// TIA Portal project "XSFW_TIA05601_A5" (V15)

(* hardware
DEVICE "S7-1200 station_1"  S7-1200 Station
   slot 0: "Rack_0"  S7-1200 Rack  Rack  V1.0
   slot 1: "PLC_1"  CPU 1214C DC/DC/DC  6ES7 214-1AG40-0XB0  V4.2
DEVICE "Dispositivo GSD_1"  GSD.Device.PN
   slot 0: "Rack"  Rack  V1.0
   slot 0: "SINAMICS-S120-CU320-2PN"  SINAMICS S120/S150 CU320-2 PN V4.7  6SL3 040-1MA01-0AAx  V4.70
      slot 0: "SINAMICS S120/S150 CU320-2 PN V4.7"  SINAMICS S120/S150 CU320-2 PN V4.7
      slot 1: "PN-IO"  PN-IO
         slot 1: "Puerto 1"  Port 1
         slot 2: "Puerto 2"  Port 2
   slot 1: "DO Control Unit_1"  DO Control Unit
      slot 0: "Punto de acceso a módulo"  Module Access Point
      slot 1: "sin PROFIsafe"  without PROFIsafe
   slot 2: "Telegrama SIEMENS 390, PZD-2/2"  SIEMENS telegram 390, PZD-2/2
   slot 2: "DO SERVO_3"  DO SERVO
      slot 0: "Punto de acceso a módulo"  Module Access Point
   slot 2: "Telegrama SIEMENS 110, PZD-12/7"  SIEMENS telegram 110, PZD-12/7
   slot 2: "Telegrama SIEMENS 370, PZD-1/1"  SIEMENS telegram 370, PZD-1/1
   slot 2: "Telegrama estándar 1, PZD-2/2"  Standard telegram 1, PZD-2/2
   slot 3: "DO Alimentación_1"  DO infeed
      slot 0: "Punto de acceso a módulo"  Module Access Point
      slot 1: "sin PROFIsafe"  without PROFIsafe
*)

// ===== PLC "PLC_1"  CPU 1214C DC/DC/DC =====

VAR_GLOBAL   // PLC tag table "Tabla de variables estándar"
   "MANDO_PLC" AT %Q72.2 : Bool;
   "System_Byte" AT %MB1 : Byte;
   "FirstScan" AT %M1.0 : Bool;
   "DiagStatusUpdate" AT %M1.1 : Bool;
   "AlwaysTRUE" AT %M1.2 : Bool;
   "AlwaysFALSE" AT %M1.3 : Bool;
   "Clock_Byte" AT %MB0 : Byte;
   "Clock_10Hz" AT %M0.0 : Bool;
   "Clock_5Hz" AT %M0.1 : Bool;
   "Clock_2.5Hz" AT %M0.2 : Bool;
   "Clock_2Hz" AT %M0.3 : Bool;
   "Clock_1.25Hz" AT %M0.4 : Bool;
   "Clock_1Hz" AT %M0.5 : Bool;
   "Clock_0.625Hz" AT %M0.6 : Bool;
   "Clock_0.5Hz" AT %M0.7 : Bool;
   "Tag_1" AT %Q64.2 : Bool;
   "Tag_2" AT %Q64.3 : Bool;
   "DES_1" AT %Q73.0 : Bool;
   "DES_2" AT %Q73.1 : Bool;
   "DES_3" AT %Q73.2 : Bool;
   "Habilito_Servicio" AT %Q73.3 : Bool;
   "Desecho_Peticion" AT %Q73.4 : Bool;
   "Parada_Intermedia" AT %Q73.5 : Bool;
   "Tag_9" AT %Q73.6 : Bool;
   "ConfirmoFallo_DRIVE" AT %Q73.7 : Bool;
   "Tag_11" AT %M10.0 : Bool;
   "Tag_12" AT %Q66.0 : Bool;
   "Activo_Contactor" AT %Q67.0 : Bool;
   "Consigna_Posicion" AT %QD82 : DWord;
   "Modo_MDI" AT %Q74.7 : Bool;
   "Correccion_Velocidad" AT %QW80 : Word;
   "Tag_3" AT %Q72.4 : Bool;
   "Tag_4" AT %M11.0 : Bool;
   "Tag_5" AT %M11.1 : Bool;
   "Tag_6" AT %M11.2 : Bool;
   "Tag_7" AT %M11.3 : Bool;
   "Tag_8" AT %M11.4 : Bool;
   "Tag_13" AT %QW88 : Word;
   "Correcion_Acel" AT %QW90 : Word;
   "Consigna_Velocidad" AT %QD86 : DWord;
   "Habilito_TrenPulsos" AT %M12.0 : Bool;
   "Reset_EntradaRapida" AT %M15.0 : Bool;
   "Sentido_Giro" AT %MD100 : DWord;
   "Frecuencia" AT %MD45 : UDInt;
   "Fallo _Activo_CU" AT %I69.3 : Bool;
   "Tag_15" AT %Q96.0 : Bool;
   "DES_1_Infeed" AT %Q97.0 : Bool;
   "DES_2_Infeed" AT %Q97.1 : Bool;
   "Mando_PLC_Infeed" AT %Q96.2 : Bool;
   "Tag_19" AT %Q97.2 : Bool;
   "Habilito_Servicio_Infeed" AT %Q97.3 : Bool;
   "Tag_18" AT %M20.0 : Bool;
   "Confirmar _fallos_IF" AT %Q97.7 : Bool;
   "Tag_16" AT %M20.1 : Bool;
   "Listo_Para_Con_Infeed" AT %I91.0 : Bool;
   "Listo_Para_Serv_Infeed" AT %I91.1 : Bool;
   "Servicio_Habilitado_Infeed" AT %I91.2 : Bool;
   "Bloqueo_Conexion_Infeed" AT %I91.6 : Bool;
   "Servicio_Infeed_Habilitado" AT %M25.0 : Bool;
   "Tag_17" AT %M25.1 : Bool;
   "Fallo_Colectico_CU" AT %I68.2 : Bool;
   "Falla_Safety_CU" AT %I68.3 : Bool;
   "Fallo_Activo_IF" AT %I91.3 : Bool;
   "Fallo_Activo_DR" AT %I77.3 : Bool;
   "Tag_20" AT %M26.0 : Bool;
   "Tag_21" AT %M26.1 : Bool;
   "Tag_22" AT %M26.2 : Bool;
   "Tag_23" AT %M26.3 : Bool;
   "Tag_24" AT %M26.4 : Bool;
   "Tag_26" AT %MW86 : Word;
   "Posicion_Real" AT %ID86 : DInt;
   "Tag_25" AT %MD30 : Real;
   "Tag_27" AT %MD34 : DWord;
   "Tag_28" AT %M26.5 : Bool;
   "PuedoSetearDES1" AT %M27.0 : Bool;
   "ConfirmoFallo_CU" AT %Q65.7 : Bool;
   "Tag_10" AT %M1000.0 : Bool;
   "Tag_29" AT %Q0.6 : Bool;
END_VAR

VAR_GLOBAL   // PLC tag table "I-O"
   "Signo" AT %I0.2 : Bool;
   "Pulsos" AT %ID1000 : DWord;
   "Alarma" AT %Q0.3 : Bool;
   "Ready" AT %Q0.4 : Bool;
   "Tag_14" AT %I0.0 : Bool;
   "Parada_Emergencia" AT %I0.4 : Bool;
   "iPul_Reset_Fallos" AT %I0.5 : Bool;
   "oLamp_Fallo" AT %Q0.5 : Bool;
END_VAR

DATA_BLOCK "Prensa_DB"   // DB4
{ S7_Optimized_Access := 'TRUE' }
VERSION : 0.1
// stored: InstanceOfName Prensa
"Prensa"
BEGIN
END_DATA_BLOCK

DATA_BLOCK "Pulsos_Acumulados"   // DB7
{ S7_Optimized_Access := 'TRUE' }
VERSION : 0.1
   VAR RETAIN
      Pulsos_Acumulados : DInt;
      Relacion_Eje_Z : LReal := 0.0965;
   END_VAR
BEGIN
END_DATA_BLOCK

// folder: System blocks/Program resources

DATA_BLOCK "IEC_Timer_0_DB"   // DB3
{ S7_Optimized_Access := 'TRUE' }
AUTHOR : Simatic
FAMILY : IEC
NAME : IEC_TMR
VERSION : 1.0
// stored: InstanceOfName IEC_TIMER
"IEC_TIMER"
BEGIN
END_DATA_BLOCK

DATA_BLOCK "IEC_Timer_0_DB_1"   // DB5
{ S7_Optimized_Access := 'TRUE' }
AUTHOR : Simatic
FAMILY : IEC
NAME : IEC_TMR
VERSION : 1.0
// stored: InstanceOfName IEC_TIMER
"IEC_TIMER"
BEGIN
END_DATA_BLOCK

DATA_BLOCK "IEC_Timer_0_DB_2"   // DB6
{ S7_Optimized_Access := 'TRUE' }
AUTHOR : Simatic
FAMILY : IEC
NAME : IEC_TMR
VERSION : 1.0
// stored: InstanceOfName IEC_TIMER
"IEC_TIMER"
BEGIN
END_DATA_BLOCK

DATA_BLOCK "IEC_Timer_0_DB_3"   // DB8
{ S7_Optimized_Access := 'TRUE' }
AUTHOR : Simatic
FAMILY : IEC
NAME : IEC_TMR
VERSION : 1.0
// stored: InstanceOfName IEC_TIMER
"IEC_TIMER"
BEGIN
END_DATA_BLOCK

// folder: (top level)

FUNCTION_BLOCK "Prensa"   // FB100, LAD
{ S7_Optimized_Access := 'TRUE' }
VERSION : 0.1
   VAR
      RangoPositivo : DInt;
      RangoNegativo : DInt;
   END_VAR
   VAR_TEMP
      Aux_Real : LReal;
      Aux_Dint : DInt;
   END_VAR
   VAR_TEMP   // added for the SCL form of the ladder/FBD networks
      _w1 : Bool;
      _w2 : Bool;
      _w3 : Bool;
      _w4 : Bool;
      _w5 : Bool;
      _w6 : Bool;
   END_VAR
BEGIN

REGION Network 1: -------------------- CONTROL CONTADOR RAPIDO--------------------------
END_REGION

REGION Network 2: Invierto el sentido de giro segun la entrada "SIGNO"
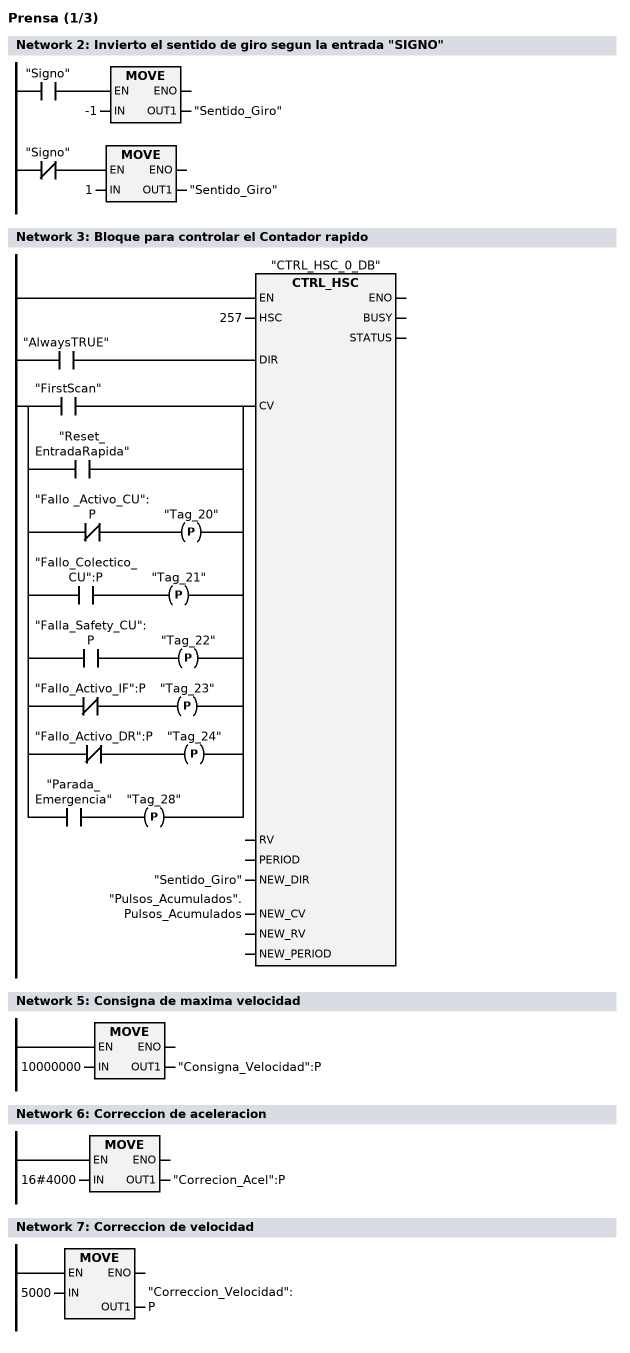
   RUNG wire#powerrail
      Contact( "Signo" )
      Move(in := -1, out1 => "Sentido_Giro")
   END_RUNG
   RUNG wire#powerrail
      I_Contact( "Signo" )
      Move(in := 1, out1 => "Sentido_Giro")
   END_RUNG
   // the same network as SCL:
   IF "Signo" THEN "Sentido_Giro" := -1; END_IF;
   IF NOT "Signo" THEN "Sentido_Giro" := 1; END_IF;
END_REGION

REGION Network 3: Bloque para controlar el Contador rapido
   #_w1 := NOT "Fallo _Activo_CU":P AND NOT "Tag_20";   // rising edge
   "Tag_20" := NOT "Fallo _Activo_CU":P;
   #_w2 := "Fallo_Colectico_CU":P AND NOT "Tag_21";   // rising edge
   "Tag_21" := "Fallo_Colectico_CU":P;
   #_w3 := "Falla_Safety_CU":P AND NOT "Tag_22";   // rising edge
   "Tag_22" := "Falla_Safety_CU":P;
   #_w4 := NOT "Fallo_Activo_IF":P AND NOT "Tag_23";   // rising edge
   "Tag_23" := NOT "Fallo_Activo_IF":P;
   #_w5 := NOT "Fallo_Activo_DR":P AND NOT "Tag_24";   // rising edge
   "Tag_24" := NOT "Fallo_Activo_DR":P;
   #_w6 := "Parada_Emergencia" AND NOT "Tag_28";   // rising edge
   "Tag_28" := "Parada_Emergencia";
   "CTRL_HSC_0_DB"(HSC := 257,   // CTRL_HSC
                   DIR := "AlwaysTRUE",
                   CV := "FirstScan" OR "Reset_EntradaRapida" OR #_w1 OR #_w2 OR #_w3 OR #_w4 OR #_w5 OR #_w6,
                   NEW_DIR := "Sentido_Giro",
                   NEW_CV := "Pulsos_Acumulados".Pulsos_Acumulados);
END_REGION

REGION Network 4: ------------------------- CONSIGNAS DE VELOCIDAD Y ACELERACION-----------------------------
END_REGION

REGION Network 5: Consigna de maxima velocidad
   RUNG wire#powerrail
      Move(in := 10000000, out1 => "Consigna_Velocidad":P)
   END_RUNG
   // the same network as SCL:
   "Consigna_Velocidad":P := 10000000;
END_REGION

REGION Network 6: Correccion de aceleracion
   RUNG wire#powerrail
      Move(in := 16#4000, out1 => "Correcion_Acel":P)
   END_RUNG
   // the same network as SCL:
   "Correcion_Acel":P := 16#4000;
END_REGION

REGION Network 7: Correccion de velocidad
   RUNG wire#powerrail
      Move(in := 5000, out1 => "Correccion_Velocidad":P)
   END_RUNG
   // the same network as SCL:
   "Correccion_Velocidad":P := 5000;
END_REGION

REGION Network 8: ---------------------------- TELEGRAMA 390------------------------
END_REGION

REGION Network 9: Telegrama 390 a Control Unit - Activo contactor
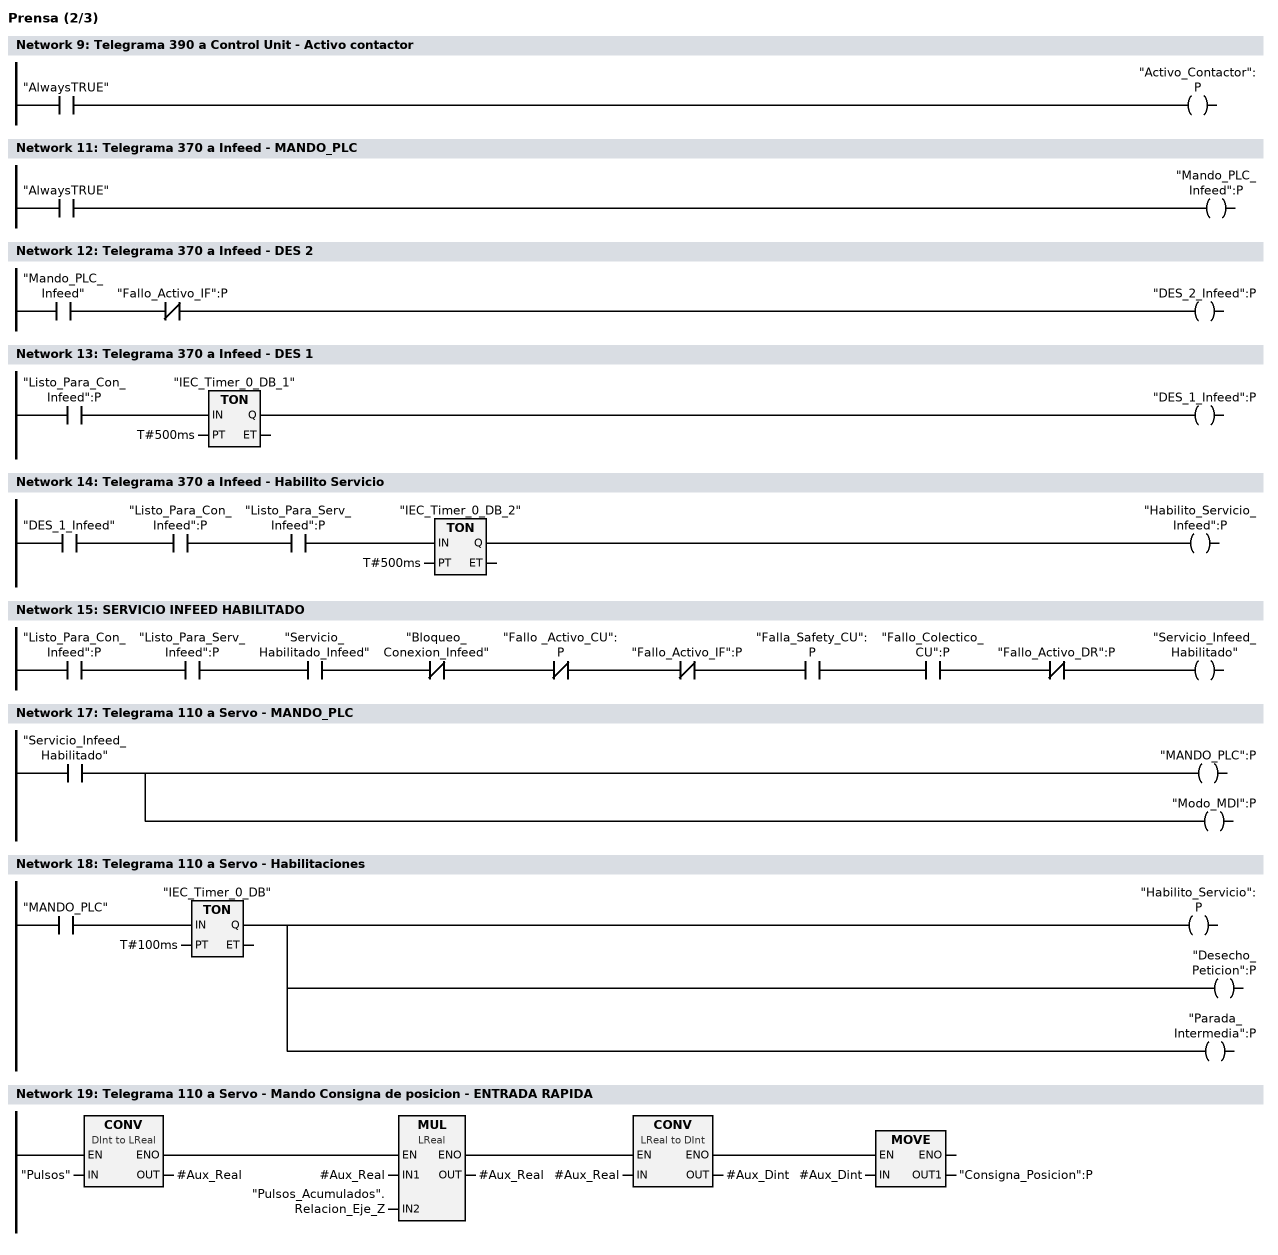
   RUNG wire#powerrail
      Contact( "AlwaysTRUE" )
      Coil( "Activo_Contactor":P )
   END_RUNG
   // the same network as SCL:
   "Activo_Contactor":P := "AlwaysTRUE";
END_REGION

REGION Network 10: ---------------------------- TELEGRAMA 370------------------------
END_REGION

REGION Network 11: Telegrama 370 a Infeed - MANDO_PLC
   RUNG wire#powerrail
      Contact( "AlwaysTRUE" )
      Coil( "Mando_PLC_Infeed":P )
   END_RUNG
   // the same network as SCL:
   "Mando_PLC_Infeed":P := "AlwaysTRUE";
END_REGION

REGION Network 12: Telegrama 370 a Infeed - DES 2
   RUNG wire#powerrail
      Contact( "Mando_PLC_Infeed" )
      I_Contact( "Fallo_Activo_IF":P )
      Coil( "DES_2_Infeed":P )
   END_RUNG
   // the same network as SCL:
   "DES_2_Infeed":P := "Mando_PLC_Infeed" AND NOT "Fallo_Activo_IF":P;
END_REGION

REGION Network 13: Telegrama 370 a Infeed - DES 1
   "IEC_Timer_0_DB_1".TON(IN := "Listo_Para_Con_Infeed":P, PT := T#500ms);
   "DES_1_Infeed":P := "IEC_Timer_0_DB_1".Q;
END_REGION

REGION Network 14: Telegrama 370 a Infeed - Habilito Servicio
   "IEC_Timer_0_DB_2".TON(IN := "DES_1_Infeed" AND "Listo_Para_Con_Infeed":P AND "Listo_Para_Serv_Infeed":P,
                          PT := T#500ms);
   "Habilito_Servicio_Infeed":P := "IEC_Timer_0_DB_2".Q;
END_REGION

REGION Network 15: SERVICIO INFEED HABILITADO
   RUNG wire#powerrail
      Contact( "Listo_Para_Con_Infeed":P )
      Contact( "Listo_Para_Serv_Infeed":P )
      Contact( "Servicio_Habilitado_Infeed" )
      I_Contact( "Bloqueo_Conexion_Infeed" )
      I_Contact( "Fallo _Activo_CU":P )
      I_Contact( "Fallo_Activo_IF":P )
      Contact( "Falla_Safety_CU":P )
      Contact( "Fallo_Colectico_CU":P )
      I_Contact( "Fallo_Activo_DR":P )
      Coil( "Servicio_Infeed_Habilitado" )
   END_RUNG
   // the same network as SCL:
   "Servicio_Infeed_Habilitado" := "Listo_Para_Con_Infeed":P AND "Listo_Para_Serv_Infeed":P AND "Servicio_Habilitado_Infeed" AND NOT "Bloqueo_Conexion_Infeed" AND NOT "Fallo _Activo_CU":P AND NOT "Fallo_Activo_IF":P AND "Falla_Safety_CU":P AND "Fallo_Colectico_CU":P AND NOT "Fallo_Activo_DR":P;
END_REGION

REGION Network 16: ---------------------------- TELEGRAMA 110------------------------
END_REGION

REGION Network 17: Telegrama 110 a Servo - MANDO_PLC
   RUNG wire#powerrail
      Contact( "Servicio_Infeed_Habilitado" )
      wire#w1
      Coil( "MANDO_PLC":P )
   END_RUNG
   RUNG wire#w1
      Coil( "Modo_MDI":P )
   END_RUNG
   // the same network as SCL:
   "MANDO_PLC":P := "Servicio_Infeed_Habilitado";
   "Modo_MDI":P := "Servicio_Infeed_Habilitado";
END_REGION

REGION Network 18: Telegrama 110 a Servo - Habilitaciones
   "IEC_Timer_0_DB".TON(IN := "MANDO_PLC", PT := T#100ms);
   "Habilito_Servicio":P := "IEC_Timer_0_DB".Q;
   "Desecho_Peticion":P := "IEC_Timer_0_DB".Q;
   "Parada_Intermedia":P := "IEC_Timer_0_DB".Q;
END_REGION

REGION Network 19: Telegrama 110 a Servo - Mando Consigna de posicion - ENTRADA RAPIDA
   RUNG wire#powerrail
      { S7_Templates := "[SrcType := DInt, DestType := LReal]" } Convert(in := "Pulsos", out => #Aux_Real)
      { S7_Templates := "SrcType := LReal" } Mul(in1 := #Aux_Real, in2 := "Pulsos_Acumulados".Relacion_Eje_Z, out => #Aux_Real)
      { S7_Templates := "[SrcType := LReal, DestType := DInt]" } Convert(in := #Aux_Real, out => #Aux_Dint)
      Move(in := #Aux_Dint, out1 => "Consigna_Posicion":P)
   END_RUNG
   // the same network as SCL:
   #Aux_Real := DINT_TO_LREAL("Pulsos");
   #Aux_Real := #Aux_Real * "Pulsos_Acumulados".Relacion_Eje_Z;
   #Aux_Dint := LREAL_TO_DINT(#Aux_Real);
   "Consigna_Posicion":P := #Aux_Dint;
END_REGION

REGION Network 20: Hiisteresis para comparar
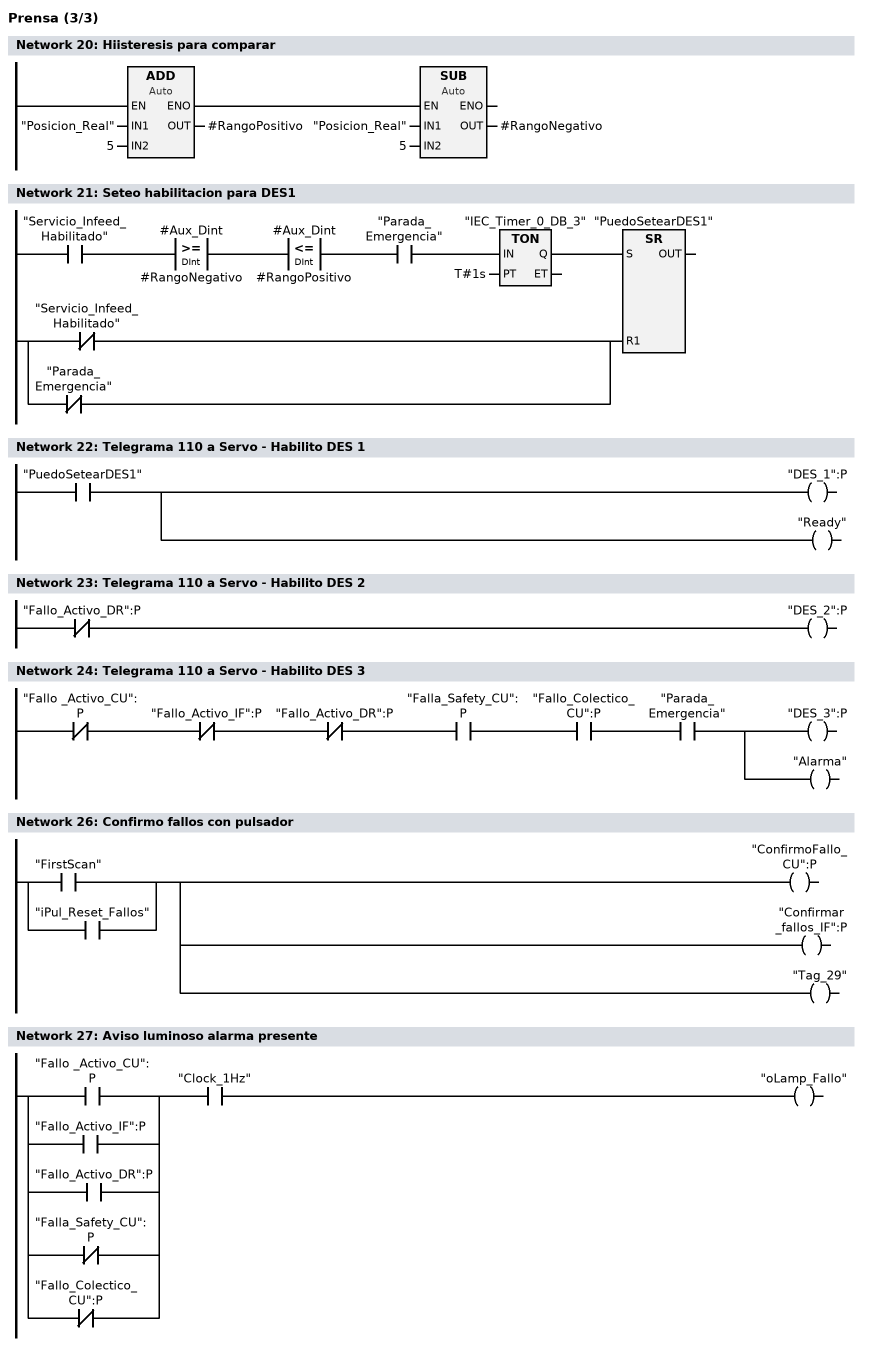
   RUNG wire#powerrail
      Add(in1 := "Posicion_Real", in2 := 5, out => #RangoPositivo)
      Sub(in1 := "Posicion_Real", in2 := 5, out => #RangoNegativo)
   END_RUNG
   // the same network as SCL:
   #RangoPositivo := "Posicion_Real" + 5;
   #RangoNegativo := "Posicion_Real" - 5;
END_REGION

REGION Network 21: Seteo habilitacion para DES1
   "IEC_Timer_0_DB_3".TON(IN := "Servicio_Infeed_Habilitado" AND (#Aux_Dint >= #RangoNegativo) AND (#Aux_Dint <= #RangoPositivo) AND "Parada_Emergencia",
                          PT := T#1s);
   IF "IEC_Timer_0_DB_3".Q THEN
       "PuedoSetearDES1" := TRUE;   // SR flip-flop
   END_IF;
   IF NOT "Servicio_Infeed_Habilitado" OR NOT "Parada_Emergencia" THEN "PuedoSetearDES1" := FALSE; END_IF;
END_REGION

REGION Network 22: Telegrama 110 a Servo - Habilito DES 1
   RUNG wire#powerrail
      Contact( "PuedoSetearDES1" )
      wire#w1
      Coil( "DES_1":P )
   END_RUNG
   RUNG wire#w1
      Coil( "Ready" )
   END_RUNG
   // the same network as SCL:
   "DES_1":P := "PuedoSetearDES1";
   "Ready" := "PuedoSetearDES1";
END_REGION

REGION Network 23: Telegrama 110 a Servo - Habilito DES 2
   RUNG wire#powerrail
      I_Contact( "Fallo_Activo_DR":P )
      Coil( "DES_2":P )
   END_RUNG
   // the same network as SCL:
   "DES_2":P := NOT "Fallo_Activo_DR":P;
END_REGION

REGION Network 24: Telegrama 110 a Servo - Habilito DES 3
   RUNG wire#powerrail
      I_Contact( "Fallo _Activo_CU":P )
      I_Contact( "Fallo_Activo_IF":P )
      I_Contact( "Fallo_Activo_DR":P )
      Contact( "Falla_Safety_CU":P )
      Contact( "Fallo_Colectico_CU":P )
      Contact( "Parada_Emergencia" )
      wire#w1
      Coil( "DES_3":P )
   END_RUNG
   RUNG wire#w1
      Coil( "Alarma" )
   END_RUNG
   // the same network as SCL:
   #_w1 := NOT "Fallo _Activo_CU":P AND NOT "Fallo_Activo_IF":P AND NOT "Fallo_Activo_DR":P AND "Falla_Safety_CU":P AND "Fallo_Colectico_CU":P AND "Parada_Emergencia";
   "DES_3":P := #_w1;
   "Alarma" := #_w1;
END_REGION

REGION Network 25: ---------------------------- CONFIRMO FALLOS ------------------------
END_REGION

REGION Network 26: Confirmo fallos con pulsador
   RUNG wire#powerrail
      Contact( "FirstScan" )
      wire#w1
      Coil( "ConfirmoFallo_CU":P )
   END_RUNG
   RUNG wire#powerrail
      Contact( "iPul_Reset_Fallos" )
   END_RUNG wire#w1
   RUNG wire#w1
      Coil( "Confirmar _fallos_IF":P )
   END_RUNG
   RUNG wire#w1
      Coil( "Tag_29" )
   END_RUNG
   // the same network as SCL:
   #_w1 := "FirstScan" OR "iPul_Reset_Fallos";
   "ConfirmoFallo_CU":P := #_w1;
   "Confirmar _fallos_IF":P := #_w1;
   "Tag_29" := #_w1;
END_REGION

REGION Network 27: Aviso luminoso alarma presente
   RUNG wire#powerrail
      Contact( "Fallo _Activo_CU":P )
      wire#w1
      Contact( "Clock_1Hz" )
      Coil( "oLamp_Fallo" )
   END_RUNG
   RUNG wire#powerrail
      Contact( "Fallo_Activo_IF":P )
   END_RUNG wire#w1
   RUNG wire#powerrail
      Contact( "Fallo_Activo_DR":P )
   END_RUNG wire#w1
   RUNG wire#powerrail
      I_Contact( "Falla_Safety_CU":P )
   END_RUNG wire#w1
   RUNG wire#powerrail
      I_Contact( "Fallo_Colectico_CU":P )
   END_RUNG wire#w1
   // the same network as SCL:
   "oLamp_Fallo" := ("Fallo _Activo_CU":P OR "Fallo_Activo_IF":P OR "Fallo_Activo_DR":P OR NOT "Falla_Safety_CU":P OR NOT "Fallo_Colectico_CU":P) AND "Clock_1Hz";
END_REGION
END_FUNCTION_BLOCK

ORGANIZATION_BLOCK "Main"   // OB1, LAD, ProgramCycle
TITLE = "Main Program Sweep (Cycle)"
{ S7_Optimized_Access := 'TRUE' }
VERSION : 0.1
   VAR_INPUT
      Initial_Call : Bool;   // Initial call of this OB
      Remanence : Bool;   // =True, if remanent data are available
   END_VAR
   VAR_TEMP
      Aux_Real : LReal;
      Aux_Dint : DInt;
   END_VAR
BEGIN

REGION Network 1: Instancia FB "Prensa"
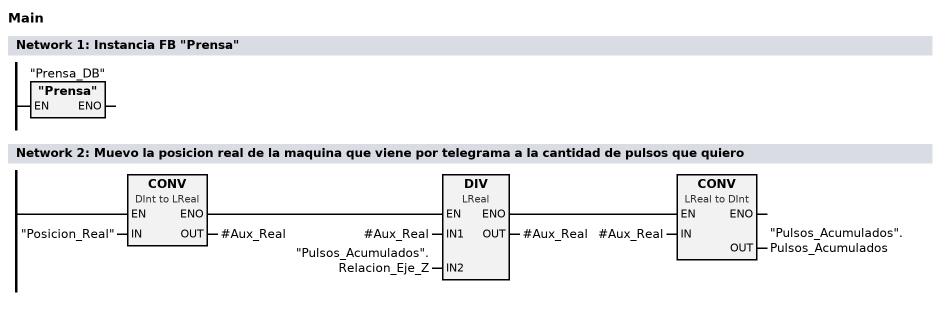
   RUNG wire#powerrail
      "Prensa_DB"()
   END_RUNG
   // the same network as SCL:
   "Prensa_DB"();   // "Prensa"
END_REGION

REGION Network 2: Muevo la posicion real de la maquina que viene por telegrama a la cantidad de pulsos que quiero
   RUNG wire#powerrail
      { S7_Templates := "[SrcType := DInt, DestType := LReal]" } Convert(in := "Posicion_Real", out => #Aux_Real)
      { S7_Templates := "SrcType := LReal" } Div(in1 := #Aux_Real, in2 := "Pulsos_Acumulados".Relacion_Eje_Z, out => #Aux_Real)
      { S7_Templates := "[SrcType := LReal, DestType := DInt]" } Convert(in := #Aux_Real, out => "Pulsos_Acumulados".Pulsos_Acumulados)
   END_RUNG
   // the same network as SCL:
   #Aux_Real := DINT_TO_LREAL("Posicion_Real");
   #Aux_Real := #Aux_Real / "Pulsos_Acumulados".Relacion_Eje_Z;
   "Pulsos_Acumulados".Pulsos_Acumulados := LREAL_TO_DINT(#Aux_Real);
END_REGION
END_ORGANIZATION_BLOCK